PROGRAM ReadAnalogInputResistance
VAR
	temp: real;
END_VAR

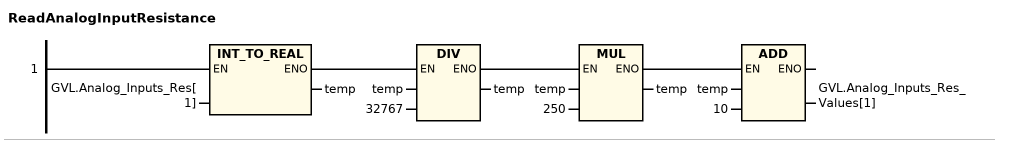
// NETWORK 1
temp := INT_TO_REAL(GVL.Analog_Inputs_Res[1]);
temp := temp / 32767;
temp := temp * 250;
GVL.Analog_Inputs_Res_Values[1] := temp + 10;

END_PROGRAM

(* stored: Version 1.1.0.1, ProductVersion 3.1.4024.12
   POU ReadAnalogInputResistance: Id {6a9fcbc0-22be-4f01-ba10-1175db0f81db}, SpecialFunc None *)
